FUNCTION_BLOCK AbfolgeTimed (* Template for a Basic Function Block Type *)
  (* Standard: 61499-2 *)
  (* Version 1.0, 2022-10-07, franz *)
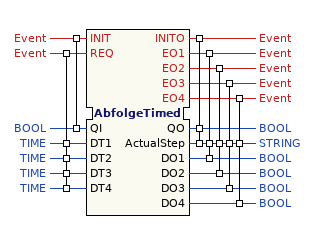
  EVENT_INPUT
    INIT WITH QI; (* Initialization Request *)
    REQ WITH DT1, DT2, DT3, DT4; (* Normal Execution Request *)
  END_EVENT
  EVENT_OUTPUT
    INITO WITH QO, ActualStep; (* Initialization Confirm *)
    EO1 WITH DO1, ActualStep;
    EO2 WITH DO2, ActualStep;
    EO3 WITH DO3, ActualStep;
    EO4 WITH DO4, ActualStep;
  END_EVENT
  VAR_INPUT
    QI : BOOL; (* Input event qualifier *)
    DT1 : TIME;
    DT2 : TIME;
    DT3 : TIME;
    DT4 : TIME;
  END_VAR
  VAR_OUTPUT
    QO : BOOL; (* Output event qualifier *)
    ActualStep : STRING;
    DO1 : BOOL;
    DO2 : BOOL;
    DO3 : BOOL;
    DO4 : BOOL;
  END_VAR
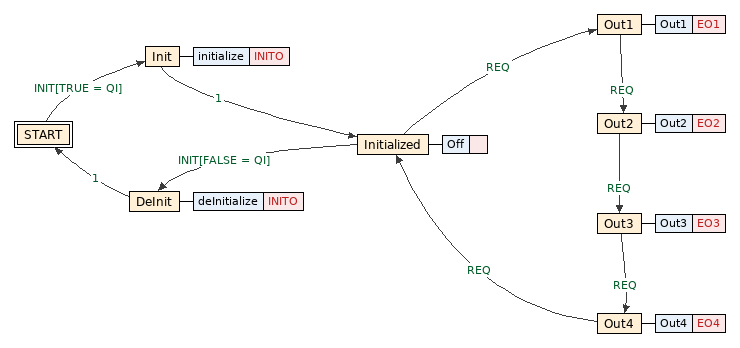
  EC_STATES
    START; (* Initial State *)
    Init : initialize -> INITO; (* Initialization *)
    Initialized : Off;
    DeInit : deInitialize -> INITO;
    Out1 : Out1 -> EO1;
    Out2 : Out2 -> EO2;
    Out3 : Out3 -> EO3;
    Out4 : Out4 -> EO4;
  END_STATES
  EC_TRANSITIONS
    START TO Init := INIT[TRUE = QI];
    Init TO Initialized := 1;
    DeInit TO START := 1;
    Initialized TO DeInit := INIT[FALSE = QI];
    Initialized TO Out1 := REQ;
    Out1 TO Out2 := REQ;
    Out2 TO Out3 := REQ;
    Out3 TO Out4 := REQ;
    Out4 TO Initialized := REQ;
  END_TRANSITIONS
  ALGORITHM initialize IN ST:
QO := QI;
ActualStep := 'initialize';
  END_ALGORITHM
  ALGORITHM deInitialize IN ST:
QO := FALSE;
ActualStep := 'deInitialize';
  END_ALGORITHM
  ALGORITHM Out1 IN ST:
DO1 := TRUE;
ActualStep := 'Out1';
  END_ALGORITHM
  ALGORITHM Out2 IN ST:
DO1 := FALSE;
DO2 := TRUE;
ActualStep := 'Out2';
  END_ALGORITHM
  ALGORITHM Out3 IN ST:
DO2 := FALSE;
DO3 := TRUE;
ActualStep := 'Out3';
  END_ALGORITHM
  ALGORITHM Out4 IN ST:
DO3 := FALSE;
DO4 := TRUE;
ActualStep := 'Out4';
  END_ALGORITHM
  ALGORITHM Off IN ST:
DO1 := FALSE;
DO2 := FALSE;
DO3 := FALSE;
DO4 := FALSE;
ActualStep := 'Off';
  END_ALGORITHM
END_FUNCTION_BLOCK
